// TIA Portal V17 export
// export: Created 2025-07-01T14:25:36.9752579Z, ExportSetting WithDefaults, DisplayName Totally Integrated Automation Portal, DisplayVersion V17 Update 8, DisplayName TIA Portal Openness, DisplayVersion V17 Update 8, DisplayName TIA Portal Version Control Interface, DisplayVersion V17, DisplayName SINAMICS Startdrive Advanced, DisplayVersion V17 SP2, DisplayName SINAMICS Startdrive G110M, G120, G120C, G120D, G120P, G115D, DisplayVersion V17 SP2, DisplayName SINAMICS Startdrive G130, G150, S120, S150, SINAMICS MV, S210, DisplayVersion V17 SP2, DisplayName STEP 7 Professional, DisplayVersion V17 Update 8, DisplayName SINUMERIK ONE STEP 7 Toolbox, DisplayVersion V17 Update 12, DisplayName SINUMERIK ONE PLC Basic Program Plus, DisplayVersion V17 Update 12, DisplayName SINUMERIK 840D sl STEP 7 Toolbox, DisplayVersion V17 Update 12, DisplayName STEP 7 Safety, DisplayVersion V17 Update 6, DisplayName WinCC Advanced, DisplayVersion V17 Update 8
FUNCTION "FC323_CHANNEL_3" : Void   // FC323, LAD
{ S7_Optimized_Access := 'FALSE' }
AUTHOR : ETXETAR
VERSION : 1.0
// stored: AutoNumber false, IsIECCheckEnabled false, SetENOAutomatically false, UDAEnableTagReadback false
   VAR_TEMP
      NC_RESET_CH3 : Bool;
      NC_START_CH3 : Bool;
   END_VAR
BEGIN

REGION Network 1: RESET CHANNEL 3
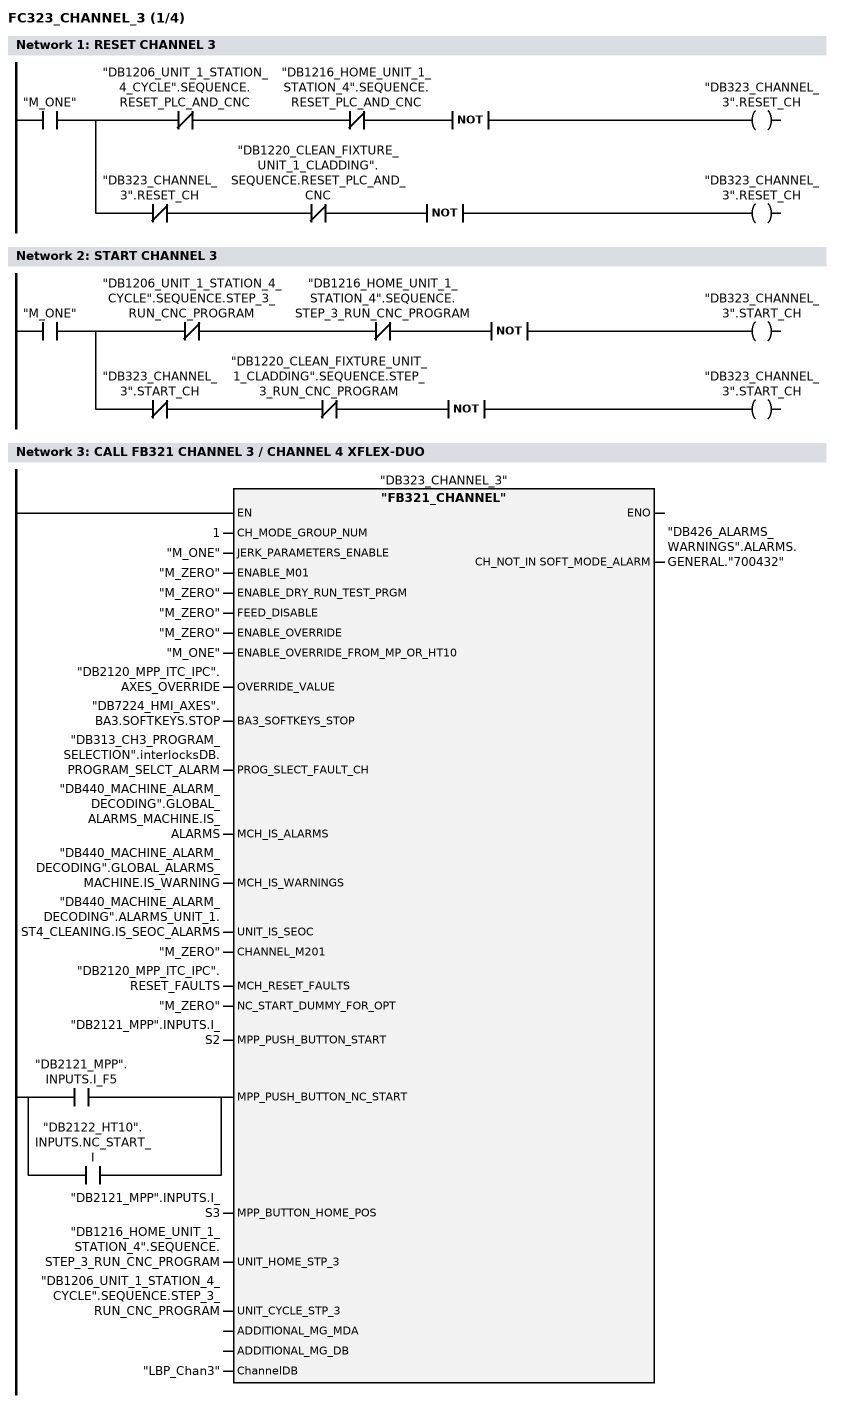
   RUNG wire#powerrail
      Contact( "M_ONE" )
      wire#w1
      I_Contact( "DB1206_UNIT_1_STATION_4_CYCLE".SEQUENCE.RESET_PLC_AND_CNC )
      I_Contact( "DB1216_HOME_UNIT_1_STATION_4".SEQUENCE.RESET_PLC_AND_CNC )
      Not()
      Coil( "DB323_CHANNEL_3".RESET_CH )
   END_RUNG
   RUNG wire#w1
      I_Contact( "DB323_CHANNEL_3".RESET_CH )
      I_Contact( "DB1220_CLEAN_FIXTURE_UNIT_1_CLADDING".SEQUENCE.RESET_PLC_AND_CNC )
      Not()
      Coil( "DB323_CHANNEL_3".RESET_CH )
   END_RUNG
   // the same network as SCL:
   "DB323_CHANNEL_3".RESET_CH := NOT ("M_ONE" AND NOT "DB1206_UNIT_1_STATION_4_CYCLE".SEQUENCE.RESET_PLC_AND_CNC AND NOT "DB1216_HOME_UNIT_1_STATION_4".SEQUENCE.RESET_PLC_AND_CNC);
   "DB323_CHANNEL_3".RESET_CH := NOT ("M_ONE" AND NOT "DB323_CHANNEL_3".RESET_CH AND NOT "DB1220_CLEAN_FIXTURE_UNIT_1_CLADDING".SEQUENCE.RESET_PLC_AND_CNC);
END_REGION

REGION Network 2: START CHANNEL 3
   RUNG wire#powerrail
      Contact( "M_ONE" )
      wire#w1
      I_Contact( "DB1206_UNIT_1_STATION_4_CYCLE".SEQUENCE.STEP_3_RUN_CNC_PROGRAM )
      I_Contact( "DB1216_HOME_UNIT_1_STATION_4".SEQUENCE.STEP_3_RUN_CNC_PROGRAM )
      Not()
      Coil( "DB323_CHANNEL_3".START_CH )
   END_RUNG
   RUNG wire#w1
      I_Contact( "DB323_CHANNEL_3".START_CH )
      I_Contact( "DB1220_CLEAN_FIXTURE_UNIT_1_CLADDING".SEQUENCE.STEP_3_RUN_CNC_PROGRAM )
      Not()
      Coil( "DB323_CHANNEL_3".START_CH )
   END_RUNG
   // the same network as SCL:
   "DB323_CHANNEL_3".START_CH := NOT ("M_ONE" AND NOT "DB1206_UNIT_1_STATION_4_CYCLE".SEQUENCE.STEP_3_RUN_CNC_PROGRAM AND NOT "DB1216_HOME_UNIT_1_STATION_4".SEQUENCE.STEP_3_RUN_CNC_PROGRAM);
   "DB323_CHANNEL_3".START_CH := NOT ("M_ONE" AND NOT "DB323_CHANNEL_3".START_CH AND NOT "DB1220_CLEAN_FIXTURE_UNIT_1_CLADDING".SEQUENCE.STEP_3_RUN_CNC_PROGRAM);
END_REGION

REGION Network 3: CALL FB321 CHANNEL 3 / CHANNEL 4 XFLEX-DUO
   RUNG wire#powerrail
      "DB323_CHANNEL_3"(MPP_PUSH_BUTTON_NC_START := wire#w1, CH_MODE_GROUP_NUM := 1, JERK_PARAMETERS_ENABLE := "M_ONE", ENABLE_M01 := "M_ZERO", ENABLE_DRY_RUN_TEST_PRGM := "M_ZERO", FEED_DISABLE := "M_ZERO", ENABLE_OVERRIDE := "M_ZERO", ENABLE_OVERRIDE_FROM_MP_OR_HT10 := "M_ONE", OVERRIDE_VALUE := "DB2120_MPP_ITC_IPC".AXES_OVERRIDE, BA3_SOFTKEYS_STOP := "DB7224_HMI_AXES".BA3.SOFTKEYS.STOP, PROG_SLECT_FAULT_CH := "DB313_CH3_PROGRAM_SELECTION".interlocksDB.PROGRAM_SELCT_ALARM, MCH_IS_ALARMS := "DB440_MACHINE_ALARM_DECODING".GLOBAL_ALARMS_MACHINE.IS_ALARMS, MCH_IS_WARNINGS := "DB440_MACHINE_ALARM_DECODING".GLOBAL_ALARMS_MACHINE.IS_WARNING, UNIT_IS_SEOC := "DB440_MACHINE_ALARM_DECODING".ALARMS_UNIT_1.ST4_CLEANING.IS_SEOC_ALARMS, CHANNEL_M201 := "M_ZERO", MCH_RESET_FAULTS := "DB2120_MPP_ITC_IPC".RESET_FAULTS, NC_START_DUMMY_FOR_OPT := "M_ZERO", MPP_PUSH_BUTTON_START := "DB2121_MPP".INPUTS.I_S2, MPP_BUTTON_HOME_POS := "DB2121_MPP".INPUTS.I_S3, UNIT_HOME_STP_3 := "DB1216_HOME_UNIT_1_STATION_4".SEQUENCE.STEP_3_RUN_CNC_PROGRAM, UNIT_CYCLE_STP_3 := "DB1206_UNIT_1_STATION_4_CYCLE".SEQUENCE.STEP_3_RUN_CNC_PROGRAM, ADDITIONAL_MG_MDA :=, ADDITIONAL_MG_DB :=, ChannelDB := "LBP_Chan3", "CH_NOT_IN SOFT_MODE_ALARM" => "DB426_ALARMS_WARNINGS".ALARMS.GENERAL."700432")
   END_RUNG
   RUNG wire#powerrail
      Contact( "DB2121_MPP".INPUTS.I_F5 )
   END_RUNG wire#w1
   RUNG wire#powerrail
      Contact( "DB2122_HT10".INPUTS.NC_START_I )
   END_RUNG wire#w1
   // the same network as SCL:
   "DB323_CHANNEL_3"(CH_MODE_GROUP_NUM := 1,   // "FB321_CHANNEL"
                     JERK_PARAMETERS_ENABLE := "M_ONE",
                     ENABLE_M01 := "M_ZERO",
                     ENABLE_DRY_RUN_TEST_PRGM := "M_ZERO",
                     FEED_DISABLE := "M_ZERO",
                     ENABLE_OVERRIDE := "M_ZERO",
                     ENABLE_OVERRIDE_FROM_MP_OR_HT10 := "M_ONE",
                     OVERRIDE_VALUE := "DB2120_MPP_ITC_IPC".AXES_OVERRIDE,
                     BA3_SOFTKEYS_STOP := "DB7224_HMI_AXES".BA3.SOFTKEYS.STOP,
                     PROG_SLECT_FAULT_CH := "DB313_CH3_PROGRAM_SELECTION".interlocksDB.PROGRAM_SELCT_ALARM,
                     MCH_IS_ALARMS := "DB440_MACHINE_ALARM_DECODING".GLOBAL_ALARMS_MACHINE.IS_ALARMS,
                     MCH_IS_WARNINGS := "DB440_MACHINE_ALARM_DECODING".GLOBAL_ALARMS_MACHINE.IS_WARNING,
                     UNIT_IS_SEOC := "DB440_MACHINE_ALARM_DECODING".ALARMS_UNIT_1.ST4_CLEANING.IS_SEOC_ALARMS,
                     CHANNEL_M201 := "M_ZERO",
                     MCH_RESET_FAULTS := "DB2120_MPP_ITC_IPC".RESET_FAULTS,
                     NC_START_DUMMY_FOR_OPT := "M_ZERO",
                     MPP_PUSH_BUTTON_START := "DB2121_MPP".INPUTS.I_S2,
                     MPP_PUSH_BUTTON_NC_START := "DB2121_MPP".INPUTS.I_F5 OR "DB2122_HT10".INPUTS.NC_START_I,
                     MPP_BUTTON_HOME_POS := "DB2121_MPP".INPUTS.I_S3,
                     UNIT_HOME_STP_3 := "DB1216_HOME_UNIT_1_STATION_4".SEQUENCE.STEP_3_RUN_CNC_PROGRAM,
                     UNIT_CYCLE_STP_3 := "DB1206_UNIT_1_STATION_4_CYCLE".SEQUENCE.STEP_3_RUN_CNC_PROGRAM,
                     ChannelDB := "LBP_Chan3",
                     "CH_NOT_IN SOFT_MODE_ALARM" => "DB426_ALARMS_WARNINGS".ALARMS.GENERAL."700432");
END_REGION

REGION Network 4: REQUEST CHANNEL 3
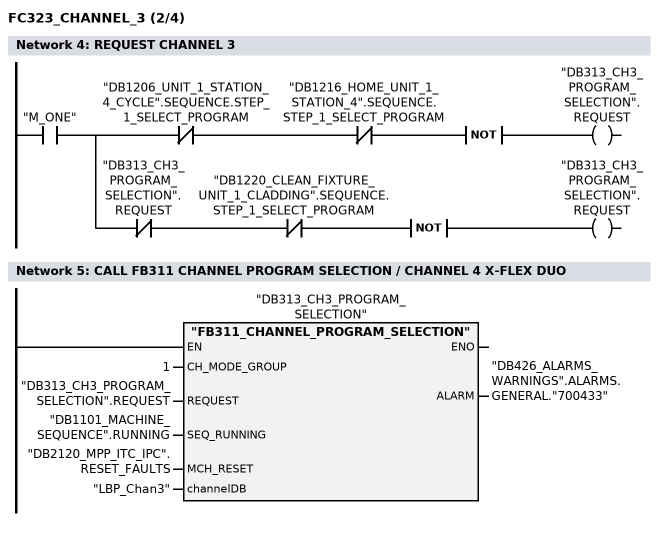
   RUNG wire#powerrail
      Contact( "M_ONE" )
      wire#w1
      I_Contact( "DB1206_UNIT_1_STATION_4_CYCLE".SEQUENCE.STEP_1_SELECT_PROGRAM )
      I_Contact( "DB1216_HOME_UNIT_1_STATION_4".SEQUENCE.STEP_1_SELECT_PROGRAM )
      Not()
      Coil( "DB313_CH3_PROGRAM_SELECTION".REQUEST )
   END_RUNG
   RUNG wire#w1
      I_Contact( "DB313_CH3_PROGRAM_SELECTION".REQUEST )
      I_Contact( "DB1220_CLEAN_FIXTURE_UNIT_1_CLADDING".SEQUENCE.STEP_1_SELECT_PROGRAM )
      Not()
      Coil( "DB313_CH3_PROGRAM_SELECTION".REQUEST )
   END_RUNG
   // the same network as SCL:
   "DB313_CH3_PROGRAM_SELECTION".REQUEST := NOT ("M_ONE" AND NOT "DB1206_UNIT_1_STATION_4_CYCLE".SEQUENCE.STEP_1_SELECT_PROGRAM AND NOT "DB1216_HOME_UNIT_1_STATION_4".SEQUENCE.STEP_1_SELECT_PROGRAM);
   "DB313_CH3_PROGRAM_SELECTION".REQUEST := NOT ("M_ONE" AND NOT "DB313_CH3_PROGRAM_SELECTION".REQUEST AND NOT "DB1220_CLEAN_FIXTURE_UNIT_1_CLADDING".SEQUENCE.STEP_1_SELECT_PROGRAM);
END_REGION

REGION Network 5: CALL FB311 CHANNEL PROGRAM SELECTION / CHANNEL 4 X-FLEX DUO
   RUNG wire#powerrail
      "DB313_CH3_PROGRAM_SELECTION"(CH_MODE_GROUP := 1, REQUEST := "DB313_CH3_PROGRAM_SELECTION".REQUEST, SEQ_RUNNING := "DB1101_MACHINE_SEQUENCE".RUNNING, MCH_RESET := "DB2120_MPP_ITC_IPC".RESET_FAULTS, channelDB := "LBP_Chan3", ALARM => "DB426_ALARMS_WARNINGS".ALARMS.GENERAL."700433")
   END_RUNG
   // the same network as SCL:
   "DB313_CH3_PROGRAM_SELECTION"(CH_MODE_GROUP := 1,   // "FB311_CHANNEL_PROGRAM_SELECTION"
                           REQUEST := "DB313_CH3_PROGRAM_SELECTION".REQUEST,
                           SEQ_RUNNING := "DB1101_MACHINE_SEQUENCE".RUNNING,
                           MCH_RESET := "DB2120_MPP_ITC_IPC".RESET_FAULTS,
                           channelDB := "LBP_Chan3",
                           ALARM => "DB426_ALARMS_WARNINGS".ALARMS.GENERAL."700433");
END_REGION

REGION Network 6: CALL FB301 CHANNEL READ AXES POSITIONS
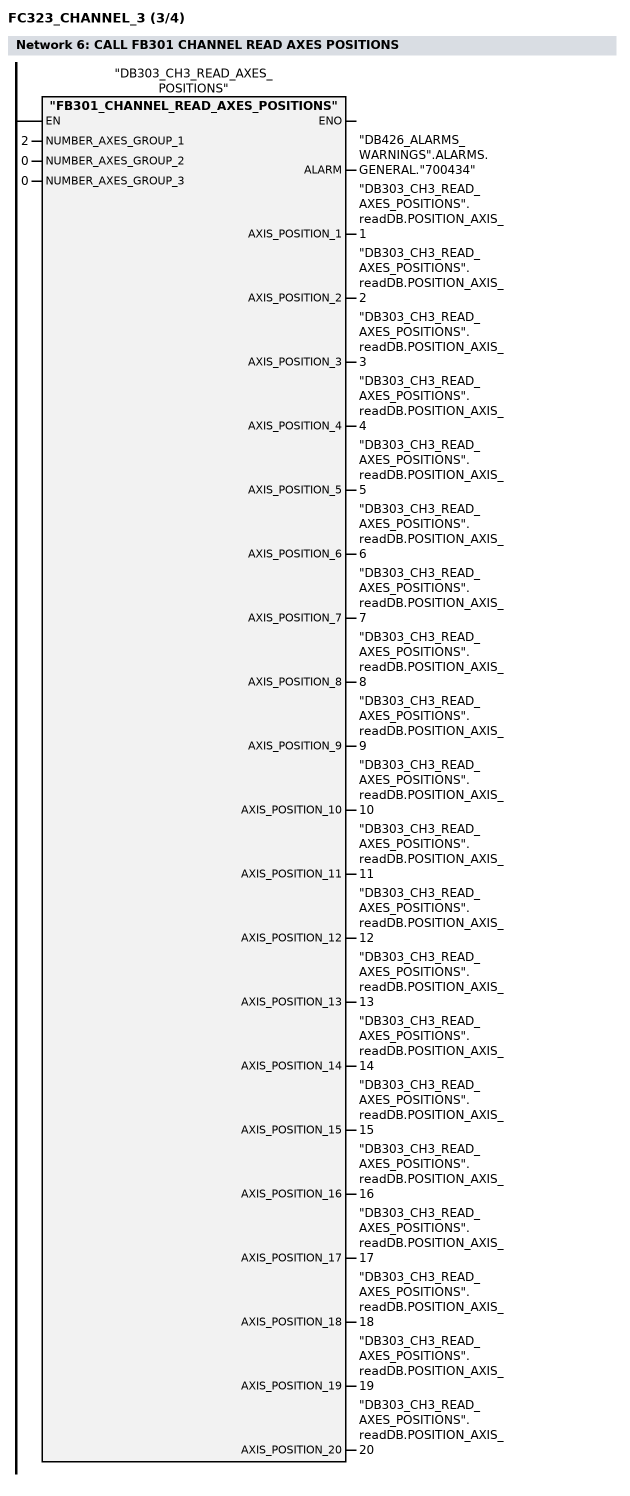
   RUNG wire#powerrail
      "DB303_CH3_READ_AXES_POSITIONS"(NUMBER_AXES_GROUP_1 := 2, NUMBER_AXES_GROUP_2 := 0, NUMBER_AXES_GROUP_3 := 0, ALARM => "DB426_ALARMS_WARNINGS".ALARMS.GENERAL."700434", AXIS_POSITION_1 => "DB303_CH3_READ_AXES_POSITIONS".readDB.POSITION_AXIS_1, AXIS_POSITION_2 => "DB303_CH3_READ_AXES_POSITIONS".readDB.POSITION_AXIS_2, AXIS_POSITION_3 => "DB303_CH3_READ_AXES_POSITIONS".readDB.POSITION_AXIS_3, AXIS_POSITION_4 => "DB303_CH3_READ_AXES_POSITIONS".readDB.POSITION_AXIS_4, AXIS_POSITION_5 => "DB303_CH3_READ_AXES_POSITIONS".readDB.POSITION_AXIS_5, AXIS_POSITION_6 => "DB303_CH3_READ_AXES_POSITIONS".readDB.POSITION_AXIS_6, AXIS_POSITION_7 => "DB303_CH3_READ_AXES_POSITIONS".readDB.POSITION_AXIS_7, AXIS_POSITION_8 => "DB303_CH3_READ_AXES_POSITIONS".readDB.POSITION_AXIS_8, AXIS_POSITION_9 => "DB303_CH3_READ_AXES_POSITIONS".readDB.POSITION_AXIS_9, AXIS_POSITION_10 => "DB303_CH3_READ_AXES_POSITIONS".readDB.POSITION_AXIS_10, AXIS_POSITION_11 => "DB303_CH3_READ_AXES_POSITIONS".readDB.POSITION_AXIS_11, AXIS_POSITION_12 => "DB303_CH3_READ_AXES_POSITIONS".readDB.POSITION_AXIS_12, AXIS_POSITION_13 => "DB303_CH3_READ_AXES_POSITIONS".readDB.POSITION_AXIS_13, AXIS_POSITION_14 => "DB303_CH3_READ_AXES_POSITIONS".readDB.POSITION_AXIS_14, AXIS_POSITION_15 => "DB303_CH3_READ_AXES_POSITIONS".readDB.POSITION_AXIS_15, AXIS_POSITION_16 => "DB303_CH3_READ_AXES_POSITIONS".readDB.POSITION_AXIS_16, AXIS_POSITION_17 => "DB303_CH3_READ_AXES_POSITIONS".readDB.POSITION_AXIS_17, AXIS_POSITION_18 => "DB303_CH3_READ_AXES_POSITIONS".readDB.POSITION_AXIS_18, AXIS_POSITION_19 => "DB303_CH3_READ_AXES_POSITIONS".readDB.POSITION_AXIS_19, AXIS_POSITION_20 => "DB303_CH3_READ_AXES_POSITIONS".readDB.POSITION_AXIS_20)
   END_RUNG
   // the same network as SCL:
   "DB303_CH3_READ_AXES_POSITIONS"(NUMBER_AXES_GROUP_1 := 2,   // "FB301_CHANNEL_READ_AXES_POSITIONS"
                           NUMBER_AXES_GROUP_2 := 0,
                           NUMBER_AXES_GROUP_3 := 0,
                           ALARM => "DB426_ALARMS_WARNINGS".ALARMS.GENERAL."700434",
                           AXIS_POSITION_1 => "DB303_CH3_READ_AXES_POSITIONS".readDB.POSITION_AXIS_1,
                           AXIS_POSITION_2 => "DB303_CH3_READ_AXES_POSITIONS".readDB.POSITION_AXIS_2,
                           AXIS_POSITION_3 => "DB303_CH3_READ_AXES_POSITIONS".readDB.POSITION_AXIS_3,
                           AXIS_POSITION_4 => "DB303_CH3_READ_AXES_POSITIONS".readDB.POSITION_AXIS_4,
                           AXIS_POSITION_5 => "DB303_CH3_READ_AXES_POSITIONS".readDB.POSITION_AXIS_5,
                           AXIS_POSITION_6 => "DB303_CH3_READ_AXES_POSITIONS".readDB.POSITION_AXIS_6,
                           AXIS_POSITION_7 => "DB303_CH3_READ_AXES_POSITIONS".readDB.POSITION_AXIS_7,
                           AXIS_POSITION_8 => "DB303_CH3_READ_AXES_POSITIONS".readDB.POSITION_AXIS_8,
                           AXIS_POSITION_9 => "DB303_CH3_READ_AXES_POSITIONS".readDB.POSITION_AXIS_9,
                           AXIS_POSITION_10 => "DB303_CH3_READ_AXES_POSITIONS".readDB.POSITION_AXIS_10,
                           AXIS_POSITION_11 => "DB303_CH3_READ_AXES_POSITIONS".readDB.POSITION_AXIS_11,
                           AXIS_POSITION_12 => "DB303_CH3_READ_AXES_POSITIONS".readDB.POSITION_AXIS_12,
                           AXIS_POSITION_13 => "DB303_CH3_READ_AXES_POSITIONS".readDB.POSITION_AXIS_13,
                           AXIS_POSITION_14 => "DB303_CH3_READ_AXES_POSITIONS".readDB.POSITION_AXIS_14,
                           AXIS_POSITION_15 => "DB303_CH3_READ_AXES_POSITIONS".readDB.POSITION_AXIS_15,
                           AXIS_POSITION_16 => "DB303_CH3_READ_AXES_POSITIONS".readDB.POSITION_AXIS_16,
                           AXIS_POSITION_17 => "DB303_CH3_READ_AXES_POSITIONS".readDB.POSITION_AXIS_17,
                           AXIS_POSITION_18 => "DB303_CH3_READ_AXES_POSITIONS".readDB.POSITION_AXIS_18,
                           AXIS_POSITION_19 => "DB303_CH3_READ_AXES_POSITIONS".readDB.POSITION_AXIS_19,
                           AXIS_POSITION_20 => "DB303_CH3_READ_AXES_POSITIONS".readDB.POSITION_AXIS_20);
END_REGION

REGION Network 7: CALL FC353 NCK M STA 4 / CALL FC1182
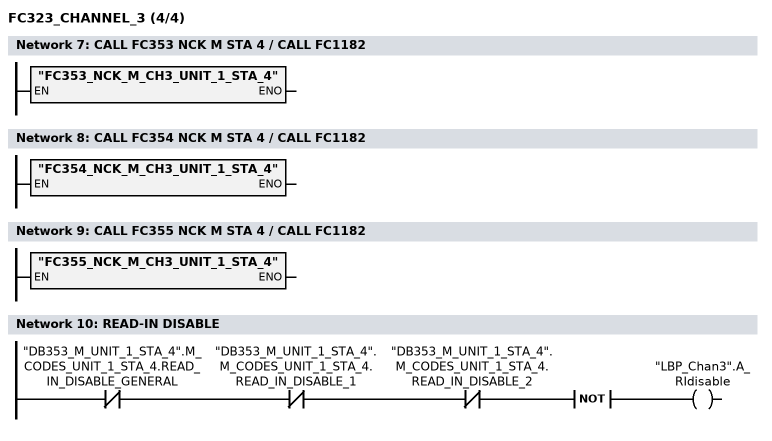
   RUNG wire#powerrail
      "FC353_NCK_M_CH3_UNIT_1_STA_4"()
   END_RUNG
   // the same network as SCL:
   "FC353_NCK_M_CH3_UNIT_1_STA_4"();
END_REGION

REGION Network 8: CALL FC354 NCK M STA 4 / CALL FC1182
   RUNG wire#powerrail
      "FC354_NCK_M_CH3_UNIT_1_STA_4"()
   END_RUNG
   // the same network as SCL:
   "FC354_NCK_M_CH3_UNIT_1_STA_4"();
END_REGION

REGION Network 9: CALL FC355 NCK M STA 4 / CALL FC1182
   RUNG wire#powerrail
      "FC355_NCK_M_CH3_UNIT_1_STA_4"()
   END_RUNG
   // the same network as SCL:
   "FC355_NCK_M_CH3_UNIT_1_STA_4"();
END_REGION

REGION Network 10: READ-IN DISABLE
   RUNG wire#powerrail
      I_Contact( "DB353_M_UNIT_1_STA_4".M_CODES_UNIT_1_STA_4.READ_IN_DISABLE_GENERAL )
      I_Contact( "DB353_M_UNIT_1_STA_4".M_CODES_UNIT_1_STA_4.READ_IN_DISABLE_1 )
      I_Contact( "DB353_M_UNIT_1_STA_4".M_CODES_UNIT_1_STA_4.READ_IN_DISABLE_2 )
      Not()
      Coil( "LBP_Chan3".A_RIdisable )
   END_RUNG
   // the same network as SCL:
   "LBP_Chan3".A_RIdisable := NOT (NOT "DB353_M_UNIT_1_STA_4".M_CODES_UNIT_1_STA_4.READ_IN_DISABLE_GENERAL AND NOT "DB353_M_UNIT_1_STA_4".M_CODES_UNIT_1_STA_4.READ_IN_DISABLE_1 AND NOT "DB353_M_UNIT_1_STA_4".M_CODES_UNIT_1_STA_4.READ_IN_DISABLE_2);
END_REGION
END_FUNCTION
